	W =  90.000 deg,	P =   0.000 deg,	R =   90.000 deg
};
P[890]{
   GP1:
	UF : 0, UT : 6,		CONFIG : 'N U T, 0, 0, 0',
	X =  218.599  mm,	Y =   -339.634  mm,	Z =   -237.572  mm,
	W =  90.000 deg,	P =   0.000 deg,	R =   90.000 deg
};
P[891]{
   GP1:
	UF : 0, UT : 6,		CONFIG : 'N U T, 0, 0, 0',
	X =  217.772  mm,	Y =   -340.100  mm,	Z =   -237.423  mm,
	W =  90.000 deg,	P =   0.000 deg,	R =   90.000 deg
};
P[892]{
   GP1:
	UF : 0, UT : 6,		CONFIG : 'N U T, 0, 0, 0',
	X =  216.761  mm,	Y =   -340.659  mm,	Z =   -237.124  mm,
	W =  90.000 deg,	P =   0.000 deg,	R =   90.000 deg
};
P[893]{
   GP1:
	UF : 0, UT : 6,		CONFIG : 'N U T, 0, 0, 0',
	X =  216.374  mm,	Y =   -340.918  mm,	Z =   -237.567  mm,
	W =  90.000 deg,	P =   0.000 deg,	R =   90.000 deg
};
P[894]{
   GP1:
	UF : 0, UT : 6,		CONFIG : 'N U T, 0, 0, 0',
	X =  212.724  mm,	Y =   -343.017  mm,	Z =   -237.456  mm,
	W =  90.000 deg,	P =   0.000 deg,	R =   90.000 deg
};
P[895]{
   GP1:
	UF : 0, UT : 6,		CONFIG : 'N U T, 0, 0, 0',
	X =  211.286  mm,	Y =   -343.853  mm,	Z =   -237.533  mm,
	W =  90.000 deg,	P =   0.000 deg,	R =   90.000 deg
};
P[896]{
   GP1:
	UF : 0, UT : 6,		CONFIG : 'N U T, 0, 0, 0',
	X =  210.442  mm,	Y =   -344.341  mm,	Z =   -237.534  mm,
	W =  90.000 deg,	P =   0.000 deg,	R =   90.000 deg
};
P[897]{
   GP1:
	UF : 0, UT : 6,		CONFIG : 'N U T, 0, 0, 0',
	X =  209.616  mm,	Y =   -344.820  mm,	Z =   -237.559  mm,
	W =  90.000 deg,	P =   0.000 deg,	R =   90.000 deg
};
P[898]{
   GP1:
	UF : 0, UT : 6,		CONFIG : 'N U T, 0, 0, 0',
	X =  209.031  mm,	Y =   -345.159  mm,	Z =   -237.581  mm,
	W =  90.000 deg,	P =   0.000 deg,	R =   90.000 deg
};
P[899]{
   GP1:
	UF : 0, UT : 6,		CONFIG : 'N U T, 0, 0, 0',
	X =  208.174  mm,	Y =   -345.643  mm,	Z =   -237.446  mm,
	W =  90.000 deg,	P =   0.000 deg,	R =   90.000 deg
};
P[900]{
   GP1:
	UF : 0, UT : 6,		CONFIG : 'N U T, 0, 0, 0',
	X =  207.552  mm,	Y =   -345.976  mm,	Z =   -237.125  mm,
	W =  90.000 deg,	P =   0.000 deg,	R =   90.000 deg
};
P[901]{
   GP1:
	UF : 0, UT : 6,		CONFIG : 'N U T, 0, 0, 0',
	X =  206.694  mm,	Y =   -346.506  mm,	Z =   -237.541  mm,
	W =  90.000 deg,	P =   0.000 deg,	R =   90.000 deg
};
P[902]{
   GP1:
	UF : 0, UT : 6,		CONFIG : 'N U T, 0, 0, 0',
	X =  205.960  mm,	Y =   -346.930  mm,	Z =   -237.542  mm,
	W =  90.000 deg,	P =   0.000 deg,	R =   90.000 deg
};
P[903]{
   GP1:
	UF : 0, UT : 6,		CONFIG : 'N U T, 0, 0, 0',
	X =  204.545  mm,	Y =   -347.747  mm,	Z =   -237.555  mm,
	W =  90.000 deg,	P =   0.000 deg,	R =   90.000 deg
};
P[904]{
   GP1:
	UF : 0, UT : 6,		CONFIG : 'N U T, 0, 0, 0',
	X =  203.611  mm,	Y =   -348.254  mm,	Z =   -237.149  mm,
	W =  90.000 deg,	P =   0.000 deg,	R =   90.000 deg
};
P[905]{
   GP1:
	UF : 0, UT : 6,		CONFIG : 'N U T, 0, 0, 0',
	X =  203.024  mm,	Y =   -348.627  mm,	Z =   -237.570  mm,
	W =  90.000 deg,	P =   0.000 deg,	R =   90.000 deg
};
P[906]{
   GP1:
	UF : 0, UT : 6,		CONFIG : 'N U T, 0, 0, 0',
	X =  201.031  mm,	Y =   -349.741  mm,	Z =   -237.128  mm,
	W =  90.000 deg,	P =   0.000 deg,	R =   90.000 deg
};
P[907]{
   GP1:
	UF : 0, UT : 6,		CONFIG : 'N U T, 0, 0, 0',
	X =  200.166  mm,	Y =   -350.274  mm,	Z =   -237.539  mm,
	W =  90.000 deg,	P =   0.000 deg,	R =   90.000 deg
};
P[908]{
   GP1:
	UF : 0, UT : 6,		CONFIG : 'N U T, 0, 0, 0',
	X =  199.491  mm,	Y =   -350.660  mm,	Z =   -237.486  mm,
	W =  90.000 deg,	P =   0.000 deg,	R =   90.000 deg
};
P[909]{
   GP1:
	UF : 0, UT : 6,		CONFIG : 'N U T, 0, 0, 0',
	X =  197.725  mm,	Y =   -351.651  mm,	Z =   -237.136  mm,
	W =  90.000 deg,	P =   0.000 deg,	R =   90.000 deg
};
P[910]{
   GP1:
	UF : 0, UT : 6,		CONFIG : 'N U T, 0, 0, 0',
	X =  196.185  mm,	Y =   -351.819  mm,	Z =   -228.207  mm,
	W =  90.000 deg,	P =   0.000 deg,	R =   90.000 deg
};
P[911]{
   GP1:
	UF : 0, UT : 6,		CONFIG : 'N U T, 0, 0, 0',
	X =  195.454  mm,	Y =   -352.239  mm,	Z =   -228.186  mm,
	W =  90.000 deg,	P =   0.000 deg,	R =   90.000 deg
};
P[912]{
   GP1:
	UF : 0, UT : 6,		CONFIG : 'N U T, 0, 0, 0',
	X =  194.680  mm,	Y =   -352.685  mm,	Z =   -228.157  mm,
	W =  90.000 deg,	P =   0.000 deg,	R =   90.000 deg
};
P[913]{
   GP1:
	UF : 0, UT : 6,		CONFIG : 'N U T, 0, 0, 0',
	X =  193.253  mm,	Y =   -353.510  mm,	Z =   -228.179  mm,
	W =  90.000 deg,	P =   0.000 deg,	R =   90.000 deg
};
P[914]{
   GP1:
	UF : 0, UT : 6,		CONFIG : 'N U T, 0, 0, 0',
	X =  190.945  mm,	Y =   -354.840  mm,	Z =   -228.146  mm,
	W =  90.000 deg,	P =   0.000 deg,	R =   90.000 deg
};
P[915]{
   GP1:
	UF : 0, UT : 6,		CONFIG : 'N U T, 0, 0, 0',
	X =  189.476  mm,	Y =   -355.695  mm,	Z =   -228.228  mm,
	W =  90.000 deg,	P =   0.000 deg,	R =   90.000 deg
};
P[916]{
   GP1:
	UF : 0, UT : 6,		CONFIG : 'N U T, 0, 0, 0',
	X =  188.747  mm,	Y =   -356.115  mm,	Z =   -228.220  mm,
	W =  90.000 deg,	P =   0.000 deg,	R =   90.000 deg
};
P[917]{
   GP1:
	UF : 0, UT : 6,		CONFIG : 'N U T, 0, 0, 0',
	X =  188.008  mm,	Y =   -356.536  mm,	Z =   -228.156  mm,
	W =  90.000 deg,	P =   0.000 deg,	R =   90.000 deg
};
P[918]{
   GP1:
	UF : 0, UT : 6,		CONFIG : 'N U T, 0, 0, 0',
	X =  187.424  mm,	Y =   -356.869  mm,	Z =   -228.099  mm,
	W =  90.000 deg,	P =   0.000 deg,	R =   90.000 deg
};
P[919]{
   GP1:
	UF : 0, UT : 6,		CONFIG : 'N U T, 0, 0, 0',
	X =  186.556  mm,	Y =   -357.376  mm,	Z =   -228.173  mm,
	W =  90.000 deg,	P =   0.000 deg,	R =   90.000 deg
};
P[920]{
   GP1:
	UF : 0, UT : 6,		CONFIG : 'N U T, 0, 0, 0',
	X =  185.070  mm,	Y =   -358.240  mm,	Z =   -228.236  mm,
	W =  90.000 deg,	P =   0.000 deg,	R =   90.000 deg
};
P[921]{
   GP1:
	UF : 0, UT : 6,		CONFIG : 'N U T, 0, 0, 0',
	X =  183.550  mm,	Y =   -359.114  mm,	Z =   -228.199  mm,
	W =  90.000 deg,	P =   0.000 deg,	R =   90.000 deg
};
P[922]{
   GP1:
	UF : 0, UT : 6,		CONFIG : 'N U T, 0, 0, 0',
	X =  182.145  mm,	Y =   -359.927  mm,	Z =   -228.216  mm,
	W =  90.000 deg,	P =   0.000 deg,	R =   90.000 deg
};
P[923]{
   GP1:
	UF : 0, UT : 6,		CONFIG : 'N U T, 0, 0, 0',
	X =  180.646  mm,	Y =   -360.783  mm,	Z =   -228.098  mm,
	W =  90.000 deg,	P =   0.000 deg,	R =   90.000 deg
};
P[924]{
   GP1:
	UF : 0, UT : 6,		CONFIG : 'N U T, 0, 0, 0',
	X =  179.919  mm,	Y =   -361.208  mm,	Z =   -228.166  mm,
	W =  90.000 deg,	P =   0.000 deg,	R =   90.000 deg
};
P[925]{
   GP1:
	UF : 0, UT : 6,		CONFIG : 'N U T, 0, 0, 0',
	X =  178.391  mm,	Y =   -362.094  mm,	Z =   -228.205  mm,
	W =  90.000 deg,	P =   0.000 deg,	R =   90.000 deg
};
P[926]{
   GP1:
	UF : 0, UT : 6,		CONFIG : 'N U T, 0, 0, 0',
	X =  177.598  mm,	Y =   -362.550  mm,	Z =   -228.194  mm,
	W =  90.000 deg,	P =   0.000 deg,	R =   90.000 deg
};
P[927]{
   GP1:
	UF : 0, UT : 6,		CONFIG : 'N U T, 0, 0, 0',
	X =  176.920  mm,	Y =   -362.944  mm,	Z =   -228.219  mm,
	W =  90.000 deg,	P =   0.000 deg,	R =   90.000 deg
};
P[928]{
   GP1:
	UF : 0, UT : 6,		CONFIG : 'N U T, 0, 0, 0',
	X =  176.225  mm,	Y =   -363.344  mm,	Z =   -228.207  mm,
	W =  90.000 deg,	P =   0.000 deg,	R =   90.000 deg
};
P[929]{
   GP1:
	UF : 0, UT : 6,		CONFIG : 'N U T, 0, 0, 0',
	X =  174.063  mm,	Y =   -364.588  mm,	Z =   -228.160  mm,
	W =  90.000 deg,	P =   0.000 deg,	R =   90.000 deg
};
P[930]{
   GP1:
	UF : 0, UT : 6,		CONFIG : 'N U T, 0, 0, 0',
	X =  172.581  mm,	Y =   -365.449  mm,	Z =   -228.218  mm,
	W =  90.000 deg,	P =   0.000 deg,	R =   90.000 deg
};
P[931]{
   GP1:
	UF : 0, UT : 6,		CONFIG : 'N U T, 0, 0, 0',
	X =  171.778  mm,	Y =   -365.897  mm,	Z =   -228.031  mm,
	W =  90.000 deg,	P =   0.000 deg,	R =   90.000 deg
};
P[932]{
   GP1:
	UF : 0, UT : 6,		CONFIG : 'N U T, 0, 0, 0',
	X =  170.454  mm,	Y =   -366.676  mm,	Z =   -228.212  mm,
	W =  90.000 deg,	P =   0.000 deg,	R =   90.000 deg
};
P[933]{
   GP1:
	UF : 0, UT : 6,		CONFIG : 'N U T, 0, 0, 0',
	X =  168.940  mm,	Y =   -367.552  mm,	Z =   -228.230  mm,
	W =  90.000 deg,	P =   0.000 deg,	R =   90.000 deg
};
P[934]{
   GP1:
	UF : 0, UT : 6,		CONFIG : 'N U T, 0, 0, 0',
	X =  168.133  mm,	Y =   -368.016  mm,	Z =   -228.209  mm,
	W =  90.000 deg,	P =   0.000 deg,	R =   90.000 deg
};
P[935]{
   GP1:
	UF : 0, UT : 6,		CONFIG : 'N U T, 0, 0, 0',
	X =  166.607  mm,	Y =   -368.891  mm,	Z =   -228.125  mm,
	W =  90.000 deg,	P =   0.000 deg,	R =   90.000 deg
};
P[936]{
   GP1:
	UF : 0, UT : 6,		CONFIG : 'N U T, 0, 0, 0',
	X =  165.799  mm,	Y =   -369.362  mm,	Z =   -228.176  mm,
	W =  90.000 deg,	P =   0.000 deg,	R =   90.000 deg
};
P[937]{
   GP1:
	UF : 0, UT : 6,		CONFIG : 'N U T, 0, 0, 0',
	X =  165.109  mm,	Y =   -369.763  mm,	Z =   -228.216  mm,
	W =  90.000 deg,	P =   0.000 deg,	R =   90.000 deg
};
P[938]{
   GP1:
	UF : 0, UT : 6,		CONFIG : 'N U T, 0, 0, 0',
	X =  164.438  mm,	Y =   -370.147  mm,	Z =   -228.169  mm,
	W =  90.000 deg,	P =   0.000 deg,	R =   90.000 deg
};
P[939]{
   GP1:
	UF : 0, UT : 6,		CONFIG : 'N U T, 0, 0, 0',
	X =  163.639  mm,	Y =   -370.610  mm,	Z =   -228.202  mm,
	W =  90.000 deg,	P =   0.000 deg,	R =   90.000 deg
};
P[940]{
   GP1:
	UF : 0, UT : 6,		CONFIG : 'N U T, 0, 0, 0',
	X =  163.129  mm,	Y =   -370.895  mm,	Z =   -228.083  mm,
	W =  90.000 deg,	P =   0.000 deg,	R =   90.000 deg
};
P[941]{
   GP1:
	UF : 0, UT : 6,		CONFIG : 'N U T, 0, 0, 0',
	X =  159.374  mm,	Y =   -373.071  mm,	Z =   -228.177  mm,
	W =  90.000 deg,	P =   0.000 deg,	R =   90.000 deg
};
P[942]{
   GP1:
	UF : 0, UT : 6,		CONFIG : 'N U T, 0, 0, 0',
	X =  157.164  mm,	Y =   -374.351  mm,	Z =   -228.219  mm,
	W =  90.000 deg,	P =   0.000 deg,	R =   90.000 deg
};
P[943]{
   GP1:
	UF : 0, UT : 6,		CONFIG : 'N U T, 0, 0, 0',
	X =  156.355  mm,	Y =   -374.816  mm,	Z =   -228.197  mm,
	W =  90.000 deg,	P =   0.000 deg,	R =   90.000 deg
};
P[944]{
   GP1:
	UF : 0, UT : 6,		CONFIG : 'N U T, 0, 0, 0',
	X =  155.638  mm,	Y =   -375.233  mm,	Z =   -228.228  mm,
	W =  90.000 deg,	P =   0.000 deg,	R =   90.000 deg
};
P[945]{
   GP1:
	UF : 0, UT : 6,		CONFIG : 'N U T, 0, 0, 0',
	X =  153.508  mm,	Y =   -376.450  mm,	Z =   -228.070  mm,
	W =  90.000 deg,	P =   0.000 deg,	R =   90.000 deg
};
P[946]{
   GP1:
	UF : 0, UT : 6,		CONFIG : 'N U T, 0, 0, 0',
	X =  151.208  mm,	Y =   -377.789  mm,	Z =   -228.208  mm,
	W =  90.000 deg,	P =   0.000 deg,	R =   90.000 deg
};
P[947]{
   GP1:
	UF : 0, UT : 6,		CONFIG : 'N U T, 0, 0, 0',
	X =  150.539  mm,	Y =   -378.176  mm,	Z =   -228.222  mm,
	W =  90.000 deg,	P =   0.000 deg,	R =   90.000 deg
};
P[948]{
   GP1:
	UF : 0, UT : 6,		CONFIG : 'N U T, 0, 0, 0',
	X =  149.740  mm,	Y =   -378.633  mm,	Z =   -228.126  mm,
	W =  90.000 deg,	P =   0.000 deg,	R =   90.000 deg
};
P[949]{
   GP1:
	UF : 0, UT : 6,		CONFIG : 'N U T, 0, 0, 0',
	X =  148.977  mm,	Y =   -379.136  mm,	Z =   -228.227  mm,
	W =  90.000 deg,	P =   0.000 deg,	R =   90.000 deg
};
P[950]{
   GP1:
	UF : 0, UT : 6,		CONFIG : 'N U T, 0, 0, 0',
	X =  148.200  mm,	Y =   -379.722  mm,	Z =   -228.031  mm,
	W =  90.000 deg,	P =   0.000 deg,	R =   90.000 deg
};
P[951]{
   GP1:
	UF : 0, UT : 6,		CONFIG : 'N U T, 0, 0, 0',
	X =  147.266  mm,	Y =   -380.698  mm,	Z =   -228.129  mm,
	W =  90.000 deg,	P =   0.000 deg,	R =   90.000 deg
};
P[952]{
   GP1:
	UF : 0, UT : 6,		CONFIG : 'N U T, 0, 0, 0',
	X =  146.233  mm,	Y =   -382.234  mm,	Z =   -228.093  mm,
	W =  90.000 deg,	P =   0.000 deg,	R =   90.000 deg
};
P[953]{
   GP1:
	UF : 0, UT : 6,		CONFIG : 'N U T, 0, 0, 0',
	X =  146.053  mm,	Y =   -382.678  mm,	Z =   -228.225  mm,
	W =  90.000 deg,	P =   0.000 deg,	R =   90.000 deg
};
P[954]{
   GP1:
	UF : 0, UT : 6,		CONFIG : 'N U T, 0, 0, 0',
	X =  145.808  mm,	Y =   -383.274  mm,	Z =   -228.209  mm,
	W =  90.000 deg,	P =   0.000 deg,	R =   90.000 deg
};
P[955]{
   GP1:
	UF : 0, UT : 6,		CONFIG : 'N U T, 0, 0, 0',
	X =  145.478  mm,	Y =   -384.435  mm,	Z =   -228.097  mm,
	W =  90.000 deg,	P =   0.000 deg,	R =   90.000 deg
};
P[956]{
   GP1:
	UF : 0, UT : 6,		CONFIG : 'N U T, 0, 0, 0',
	X =  145.381  mm,	Y =   -387.073  mm,	Z =   -228.188  mm,
	W =  90.000 deg,	P =   0.000 deg,	R =   90.000 deg
};
P[957]{
   GP1:
	UF : 0, UT : 6,		CONFIG : 'N U T, 0, 0, 0',
	X =  145.443  mm,	Y =   -387.440  mm,	Z =   -228.189  mm,
	W =  90.000 deg,	P =   0.000 deg,	R =   90.000 deg
};
P[958]{
   GP1:
	UF : 0, UT : 6,		CONFIG : 'N U T, 0, 0, 0',
	X =  146.144  mm,	Y =   -389.710  mm,	Z =   -228.125  mm,
	W =  90.000 deg,	P =   0.000 deg,	R =   90.000 deg
};
P[959]{
   GP1:
	UF : 0, UT : 6,		CONFIG : 'N U T, 0, 0, 0',
	X =  146.550  mm,	Y =   -390.502  mm,	Z =   -228.144  mm,
	W =  90.000 deg,	P =   0.000 deg,	R =   90.000 deg
};
P[960]{
   GP1:
	UF : 0, UT : 6,		CONFIG : 'N U T, 0, 0, 0',
	X =  146.942  mm,	Y =   -391.181  mm,	Z =   -228.187  mm,
	W =  90.000 deg,	P =   0.000 deg,	R =   90.000 deg
};
P[961]{
   GP1:
	UF : 0, UT : 6,		CONFIG : 'N U T, 0, 0, 0',
	X =  147.804  mm,	Y =   -392.671  mm,	Z =   -228.212  mm,
	W =  90.000 deg,	P =   0.000 deg,	R =   90.000 deg
};
P[962]{
   GP1:
	UF : 0, UT : 6,		CONFIG : 'N U T, 0, 0, 0',
	X =  148.260  mm,	Y =   -393.458  mm,	Z =   -228.223  mm,
	W =  90.000 deg,	P =   0.000 deg,	R =   90.000 deg
};
P[963]{
   GP1:
	UF : 0, UT : 6,		CONFIG : 'N U T, 0, 0, 0',
	X =  150.818  mm,	Y =   -397.896  mm,	Z =   -228.169  mm,
	W =  90.000 deg,	P =   0.000 deg,	R =   90.000 deg
};
P[964]{
   GP1:
	UF : 0, UT : 6,		CONFIG : 'N U T, 0, 0, 0',
	X =  151.256  mm,	Y =   -398.648  mm,	Z =   -228.215  mm,
	W =  90.000 deg,	P =   0.000 deg,	R =   90.000 deg
};
P[965]{
   GP1:
	UF : 0, UT : 6,		CONFIG : 'N U T, 0, 0, 0',
	X =  151.642  mm,	Y =   -399.327  mm,	Z =   -228.140  mm,
	W =  90.000 deg,	P =   0.000 deg,	R =   90.000 deg
};
P[966]{
   GP1:
	UF : 0, UT : 6,		CONFIG : 'N U T, 0, 0, 0',
	X =  153.792  mm,	Y =   -403.044  mm,	Z =   -228.191  mm,
	W =  90.000 deg,	P =   0.000 deg,	R =   90.000 deg
};
P[967]{
   GP1:
	UF : 0, UT : 6,		CONFIG : 'N U T, 0, 0, 0',
	X =  154.199  mm,	Y =   -403.752  mm,	Z =   -228.164  mm,
	W =  90.000 deg,	P =   0.000 deg,	R =   90.000 deg
};
P[968]{
   GP1:
	UF : 0, UT : 6,		CONFIG : 'N U T, 0, 0, 0',
	X =  154.648  mm,	Y =   -404.525  mm,	Z =   -228.193  mm,
	W =  90.000 deg,	P =   0.000 deg,	R =   90.000 deg
};
P[969]{
   GP1:
	UF : 0, UT : 6,		CONFIG : 'N U T, 0, 0, 0',
	X =  155.420  mm,	Y =   -405.865  mm,	Z =   -228.172  mm,
	W =  90.000 deg,	P =   0.000 deg,	R =   90.000 deg
};
P[970]{
   GP1:
	UF : 0, UT : 6,		CONFIG : 'N U T, 0, 0, 0',
	X =  155.841  mm,	Y =   -406.599  mm,	Z =   -228.138  mm,
	W =  90.000 deg,	P =   0.000 deg,	R =   90.000 deg
};
P[971]{
   GP1:
	UF : 0, UT : 6,		CONFIG : 'N U T, 0, 0, 0',
	X =  157.126  mm,	Y =   -408.820  mm,	Z =   -228.166  mm,
	W =  90.000 deg,	P =   0.000 deg,	R =   90.000 deg
};
P[972]{
   GP1:
	UF : 0, UT : 6,		CONFIG : 'N U T, 0, 0, 0',
	X =  158.080  mm,	Y =   -410.465  mm,	Z =   -228.218  mm,
	W =  90.000 deg,	P =   0.000 deg,	R =   90.000 deg
};
P[973]{
   GP1:
	UF : 0, UT : 6,		CONFIG : 'N U T, 0, 0, 0',
	X =  158.486  mm,	Y =   -411.171  mm,	Z =   -228.203  mm,
	W =  90.000 deg,	P =   0.000 deg,	R =   90.000 deg
};
P[974]{
   GP1:
	UF : 0, UT : 6,		CONFIG : 'N U T, 0, 0, 0',
	X =  158.921  mm,	Y =   -411.930  mm,	Z =   -228.164  mm,
	W =  90.000 deg,	P =   0.000 deg,	R =   90.000 deg
};
P[975]{
   GP1:
	UF : 0, UT : 6,		CONFIG : 'N U T, 0, 0, 0',
	X =  159.712  mm,	Y =   -413.295  mm,	Z =   -228.196  mm,
	W =  90.000 deg,	P =   0.000 deg,	R =   90.000 deg
};
P[976]{
   GP1:
	UF : 0, UT : 6,		CONFIG : 'N U T, 0, 0, 0',
	X =  160.187  mm,	Y =   -414.120  mm,	Z =   -228.194  mm,
	W =  90.000 deg,	P =   0.000 deg,	R =   90.000 deg
};
P[977]{
   GP1:
	UF : 0, UT : 6,		CONFIG : 'N U T, 0, 0, 0',
	X =  160.929  mm,	Y =   -415.417  mm,	Z =   -228.106  mm,
	W =  90.000 deg,	P =   0.000 deg,	R =   90.000 deg
};
P[978]{
   GP1:
	UF : 0, UT : 6,		CONFIG : 'N U T, 0, 0, 0',
	X =  161.858  mm,	Y =   -417.021  mm,	Z =   -228.139  mm,
	W =  90.000 deg,	P =   0.000 deg,	R =   90.000 deg
};
P[979]{
   GP1:
	UF : 0, UT : 6,		CONFIG : 'N U T, 0, 0, 0',
	X =  162.280  mm,	Y =   -417.744  mm,	Z =   -228.199  mm,
	W =  90.000 deg,	P =   0.000 deg,	R =   90.000 deg
};
P[980]{
   GP1:
	UF : 0, UT : 6,		CONFIG : 'N U T, 0, 0, 0',
	X =  162.737  mm,	Y =   -418.529  mm,	Z =   -228.230  mm,
	W =  90.000 deg,	P =   0.000 deg,	R =   90.000 deg
};
P[981]{
   GP1:
	UF : 0, UT : 6,		CONFIG : 'N U T, 0, 0, 0',
	X =  163.999  mm,	Y =   -420.714  mm,	Z =   -228.237  mm,
	W =  90.000 deg,	P =   0.000 deg,	R =   90.000 deg
};
P[982]{
   GP1:
	UF : 0, UT : 6,		CONFIG : 'N U T, 0, 0, 0',
	X =  164.809  mm,	Y =   -422.113  mm,	Z =   -228.236  mm,
	W =  90.000 deg,	P =   0.000 deg,	R =   90.000 deg
};
P[983]{
   GP1:
	UF : 0, UT : 6,		CONFIG : 'N U T, 0, 0, 0',
	X =  165.316  mm,	Y =   -422.912  mm,	Z =   -228.180  mm,
	W =  90.000 deg,	P =   0.000 deg,	R =   90.000 deg
};
P[984]{
   GP1:
	UF : 0, UT : 6,		CONFIG : 'N U T, 0, 0, 0',
	X =  165.883  mm,	Y =   -423.661  mm,	Z =   -228.126  mm,
	W =  90.000 deg,	P =   0.000 deg,	R =   90.000 deg
};
P[985]{
   GP1:
	UF : 0, UT : 6,		CONFIG : 'N U T, 0, 0, 0',
	X =  167.143  mm,	Y =   -424.844  mm,	Z =   -228.228  mm,
	W =  90.000 deg,	P =   0.000 deg,	R =   90.000 deg
};
P[986]{
   GP1:
	UF : 0, UT : 6,		CONFIG : 'N U T, 0, 0, 0',
	X =  167.963  mm,	Y =   -425.401  mm,	Z =   -228.187  mm,
	W =  90.000 deg,	P =   0.000 deg,	R =   90.000 deg
};
P[987]{
   GP1:
	UF : 0, UT : 6,		CONFIG : 'N U T, 0, 0, 0',
	X =  169.627  mm,	Y =   -426.176  mm,	Z =   -228.220  mm,
	W =  90.000 deg,	P =   0.000 deg,	R =   90.000 deg
};
P[988]{
   GP1:
	UF : 0, UT : 6,		CONFIG : 'N U T, 0, 0, 0',
	X =  171.276  mm,	Y =   -426.533  mm,	Z =   -228.200  mm,
	W =  90.000 deg,	P =   0.000 deg,	R =   90.000 deg
};
P[989]{
   GP1:
	UF : 0, UT : 6,		CONFIG : 'N U T, 0, 0, 0',
	X =  173.180  mm,	Y =   -426.560  mm,	Z =   -228.200  mm,
	W =  90.000 deg,	P =   0.000 deg,	R =   90.000 deg
};
P[990]{
   GP1:
	UF : 0, UT : 6,		CONFIG : 'N U T, 0, 0, 0',
	X =  174.290  mm,	Y =   -426.355  mm,	Z =   -228.235  mm,
	W =  90.000 deg,	P =   0.000 deg,	R =   90.000 deg
};
P[991]{
   GP1:
	UF : 0, UT : 6,		CONFIG : 'N U T, 0, 0, 0',
	X =  176.020  mm,	Y =   -425.728  mm,	Z =   -228.224  mm,
	W =  90.000 deg,	P =   0.000 deg,	R =   90.000 deg
};
P[992]{
   GP1:
	UF : 0, UT : 6,		CONFIG : 'N U T, 0, 0, 0',
	X =  176.814  mm,	Y =   -425.317  mm,	Z =   -228.224  mm,
	W =  90.000 deg,	P =   0.000 deg,	R =   90.000 deg
};
P[993]{
   GP1:
	UF : 0, UT : 6,		CONFIG : 'N U T, 0, 0, 0',
	X =  179.687  mm,	Y =   -423.666  mm,	Z =   -228.132  mm,
	W =  90.000 deg,	P =   0.000 deg,	R =   90.000 deg
};
P[994]{
   GP1:
	UF : 0, UT : 6,		CONFIG : 'N U T, 0, 0, 0',
	X =  181.001  mm,	Y =   -422.898  mm,	Z =   -228.235  mm,
	W =  90.000 deg,	P =   0.000 deg,	R =   90.000 deg
};
P[995]{
   GP1:
	UF : 0, UT : 6,		CONFIG : 'N U T, 0, 0, 0',
	X =  183.357  mm,	Y =   -421.546  mm,	Z =   -228.150  mm,
	W =  90.000 deg,	P =   0.000 deg,	R =   90.000 deg
};
P[996]{
   GP1:
	UF : 0, UT : 6,		CONFIG : 'N U T, 0, 0, 0',
	X =  184.091  mm,	Y =   -421.118  mm,	Z =   -228.196  mm,
	W =  90.000 deg,	P =   0.000 deg,	R =   90.000 deg
};
P[997]{
   GP1:
	UF : 0, UT : 6,		CONFIG : 'N U T, 0, 0, 0',
	X =  184.898  mm,	Y =   -420.658  mm,	Z =   -228.123  mm,
	W =  90.000 deg,	P =   0.000 deg,	R =   90.000 deg
};
P[998]{
   GP1:
	UF : 0, UT : 6,		CONFIG : 'N U T, 0, 0, 0',
	X =  186.356  mm,	Y =   -419.822  mm,	Z =   -228.052  mm,
	W =  90.000 deg,	P =   0.000 deg,	R =   90.000 deg
};
P[999]{
   GP1:
	UF : 0, UT : 6,		CONFIG : 'N U T, 0, 0, 0',
	X =  187.838  mm,	Y =   -418.954  mm,	Z =   -228.196  mm,
	W =  90.000 deg,	P =   0.000 deg,	R =   90.000 deg
};
P[1000]{
   GP1:
	UF : 0, UT : 6,		CONFIG : 'N U T, 0, 0, 0',
	X =  189.967  mm,	Y =   -417.730  mm,	Z =   -228.127  mm,
	W =  90.000 deg,	P =   0.000 deg,	R =   90.000 deg
};
P[1001]{
   GP1:
	UF : 0, UT : 6,		CONFIG : 'N U T, 0, 0, 0',
	X =  190.703  mm,	Y =   -417.300  mm,	Z =   -228.188  mm,
	W =  90.000 deg,	P =   0.000 deg,	R =   90.000 deg
};
P[1002]{
   GP1:
	UF : 0, UT : 6,		CONFIG : 'N U T, 0, 0, 0',
	X =  192.914  mm,	Y =   -416.029  mm,	Z =   -228.126  mm,
	W =  90.000 deg,	P =   0.000 deg,	R =   90.000 deg
};
P[1003]{
   GP1:
	UF : 0, UT : 6,		CONFIG : 'N U T, 0, 0, 0',
	X =  193.613  mm,	Y =   -415.619  mm,	Z =   -228.212  mm,
	W =  90.000 deg,	P =   0.000 deg,	R =   90.000 deg
};
P[1004]{
   GP1:
	UF : 0, UT : 6,		CONFIG : 'N U T, 0, 0, 0',
	X =  195.788  mm,	Y =   -414.368  mm,	Z =   -228.146  mm,
	W =  90.000 deg,	P =   0.000 deg,	R =   90.000 deg
};
P[1005]{
   GP1:
	UF : 0, UT : 6,		CONFIG : 'N U T, 0, 0, 0',
	X =  196.586  mm,	Y =   -413.902  mm,	Z =   -228.215  mm,
	W =  90.000 deg,	P =   0.000 deg,	R =   90.000 deg
};
P[1006]{
   GP1:
	UF : 0, UT : 6,		CONFIG : 'N U T, 0, 0, 0',
	X =  197.412  mm,	Y =   -413.423  mm,	Z =   -228.237  mm,
	W =  90.000 deg,	P =   0.000 deg,	R =   90.000 deg
};
P[1007]{
   GP1:
	UF : 0, UT : 6,		CONFIG : 'N U T, 0, 0, 0',
	X =  198.036  mm,	Y =   -413.064  mm,	Z =   -228.228  mm,
	W =  90.000 deg,	P =   0.000 deg,	R =   90.000 deg
};
P[1008]{
   GP1:
	UF : 0, UT : 6,		CONFIG : 'N U T, 0, 0, 0',
	X =  198.778  mm,	Y =   -412.636  mm,	Z =   -228.213  mm,
	W =  90.000 deg,	P =   0.000 deg,	R =   90.000 deg
};
P[1009]{
   GP1:
	UF : 0, UT : 6,		CONFIG : 'N U T, 0, 0, 0',
	X =  200.334  mm,	Y =   -411.737  mm,	Z =   -228.222  mm,
	W =  90.000 deg,	P =   0.000 deg,	R =   90.000 deg
};
P[1010]{
   GP1:
	UF : 0, UT : 6,		CONFIG : 'N U T, 0, 0, 0',
	X =  201.879  mm,	Y =   -410.844  mm,	Z =   -228.237  mm,
	W =  90.000 deg,	P =   0.000 deg,	R =   90.000 deg
};
P[1011]{
   GP1:
	UF : 0, UT : 6,		CONFIG : 'N U T, 0, 0, 0',
	X =  203.269  mm,	Y =   -410.050  mm,	Z =   -228.131  mm,
	W =  90.000 deg,	P =   0.000 deg,	R =   90.000 deg
};
P[1012]{
   GP1:
	UF : 0, UT : 6,		CONFIG : 'N U T, 0, 0, 0',
	X =  205.460  mm,	Y =   -408.780  mm,	Z =   -228.192  mm,
	W =  90.000 deg,	P =   0.000 deg,	R =   90.000 deg
};
P[1013]{
   GP1:
	UF : 0, UT : 6,		CONFIG : 'N U T, 0, 0, 0',
	X =  207.024  mm,	Y =   -407.878  mm,	Z =   -228.181  mm,
	W =  90.000 deg,	P =   0.000 deg,	R =   90.000 deg
};
P[1014]{
   GP1:
	UF : 0, UT : 6,		CONFIG : 'N U T, 0, 0, 0',
	X =  207.746  mm,	Y =   -407.462  mm,	Z =   -228.164  mm,
	W =  90.000 deg,	P =   0.000 deg,	R =   90.000 deg
};
P[1015]{
   GP1:
	UF : 0, UT : 6,		CONFIG : 'N U T, 0, 0, 0',
	X =  209.153  mm,	Y =   -406.651  mm,	Z =   -228.155  mm,
	W =  90.000 deg,	P =   0.000 deg,	R =   90.000 deg
};
P[1016]{
   GP1:
	UF : 0, UT : 6,		CONFIG : 'N U T, 0, 0, 0',
	X =  209.719  mm,	Y =   -406.319  mm,	Z =   -228.208  mm,
	W =  90.000 deg,	P =   0.000 deg,	R =   90.000 deg
};
P[1017]{
   GP1:
	UF : 0, UT : 6,		CONFIG : 'N U T, 0, 0, 0',
	X =  210.677  mm,	Y =   -405.769  mm,	Z =   -228.179  mm,
	W =  90.000 deg,	P =   0.000 deg,	R =   90.000 deg
};
P[1018]{
   GP1:
	UF : 0, UT : 6,		CONFIG : 'N U T, 0, 0, 0',
	X =  211.948  mm,	Y =   -405.031  mm,	Z =   -228.216  mm,
	W =  90.000 deg,	P =   0.000 deg,	R =   90.000 deg
};
P[1019]{
   GP1:
	UF : 0, UT : 6,		CONFIG : 'N U T, 0, 0, 0',
	X =  212.682  mm,	Y =   -404.610  mm,	Z =   -228.190  mm,
	W =  90.000 deg,	P =   0.000 deg,	R =   90.000 deg
};
P[1020]{
   GP1:
	UF : 0, UT : 6,		CONFIG : 'N U T, 0, 0, 0',
	X =  213.487  mm,	Y =   -404.144  mm,	Z =   -228.213  mm,
	W =  90.000 deg,	P =   0.000 deg,	R =   90.000 deg
};
P[1021]{
   GP1:
	UF : 0, UT : 6,		CONFIG : 'N U T, 0, 0, 0',
	X =  215.022  mm,	Y =   -403.262  mm,	Z =   -228.154  mm,
	W =  90.000 deg,	P =   0.000 deg,	R =   90.000 deg
};
P[1022]{
   GP1:
	UF : 0, UT : 6,		CONFIG : 'N U T, 0, 0, 0',
	X =  217.268  mm,	Y =   -401.964  mm,	Z =   -228.169  mm,
	W =  90.000 deg,	P =   0.000 deg,	R =   90.000 deg
};
P[1023]{
   GP1:
	UF : 0, UT : 6,		CONFIG : 'N U T, 0, 0, 0',
	X =  218.082  mm,	Y =   -401.493  mm,	Z =   -228.173  mm,
	W =  90.000 deg,	P =   0.000 deg,	R =   90.000 deg
};
P[1024]{
   GP1:
	UF : 0, UT : 6,		CONFIG : 'N U T, 0, 0, 0',
	X =  218.710  mm,	Y =   -401.132  mm,	Z =   -228.160  mm,
	W =  90.000 deg,	P =   0.000 deg,	R =   90.000 deg
};
P[1025]{
   GP1:
	UF : 0, UT : 6,		CONFIG : 'N U T, 0, 0, 0',
	X =  219.417  mm,	Y =   -400.722  mm,	Z =   -228.177  mm,
	W =  90.000 deg,	P =   0.000 deg,	R =   90.000 deg
};
P[1026]{
   GP1:
	UF : 0, UT : 6,		CONFIG : 'N U T, 0, 0, 0',
	X =  220.998  mm,	Y =   -399.808  mm,	Z =   -228.202  mm,
	W =  90.000 deg,	P =   0.000 deg,	R =   90.000 deg
};
P[1027]{
   GP1:
	UF : 0, UT : 6,		CONFIG : 'N U T, 0, 0, 0',
	X =  222.414  mm,	Y =   -398.991  mm,	Z =   -228.190  mm,
	W =  90.000 deg,	P =   0.000 deg,	R =   90.000 deg
};
P[1028]{
   GP1:
	UF : 0, UT : 6,		CONFIG : 'N U T, 0, 0, 0',
	X =  223.201  mm,	Y =   -398.535  mm,	Z =   -228.206  mm,
	W =  90.000 deg,	P =   0.000 deg,	R =   90.000 deg
};
P[1029]{
   GP1:
	UF : 0, UT : 6,		CONFIG : 'N U T, 0, 0, 0',
	X =  223.860  mm,	Y =   -398.162  mm,	Z =   -228.118  mm,
	W =  90.000 deg,	P =   0.000 deg,	R =   90.000 deg
};
P[1030]{
   GP1:
	UF : 0, UT : 6,		CONFIG : 'N U T, 0, 0, 0',
	X =  224.610  mm,	Y =   -397.722  mm,	Z =   -228.204  mm,
	W =  90.000 deg,	P =   0.000 deg,	R =   90.000 deg
};
P[1031]{
   GP1:
	UF : 0, UT : 6,		CONFIG : 'N U T, 0, 0, 0',
	X =  225.370  mm,	Y =   -397.282  mm,	Z =   -228.218  mm,
	W =  90.000 deg,	P =   0.000 deg,	R =   90.000 deg
};
P[1032]{
   GP1:
	UF : 0, UT : 6,		CONFIG : 'N U T, 0, 0, 0',
	X =  226.172  mm,	Y =   -396.828  mm,	Z =   -228.106  mm,
	W =  90.000 deg,	P =   0.000 deg,	R =   90.000 deg
};
P[1033]{
   GP1:
	UF : 0, UT : 6,		CONFIG : 'N U T, 0, 0, 0',
	X =  226.816  mm,	Y =   -396.457  mm,	Z =   -228.097  mm,
	W =  90.000 deg,	P =   0.000 deg,	R =   90.000 deg
};
P[1034]{
   GP1:
	UF : 0, UT : 6,		CONFIG : 'N U T, 0, 0, 0',
	X =  228.225  mm,	Y =   -395.635  mm,	Z =   -228.203  mm,
	W =  90.000 deg,	P =   0.000 deg,	R =   90.000 deg
};
P[1035]{
   GP1:
	UF : 0, UT : 6,		CONFIG : 'N U T, 0, 0, 0',
	X =  229.019  mm,	Y =   -395.182  mm,	Z =   -228.134  mm,
	W =  90.000 deg,	P =   0.000 deg,	R =   90.000 deg
};
P[1036]{
   GP1:
	UF : 0, UT : 6,		CONFIG : 'N U T, 0, 0, 0',
	X =  232.005  mm,	Y =   -393.450  mm,	Z =   -228.230  mm,
	W =  90.000 deg,	P =   0.000 deg,	R =   90.000 deg
};
P[1037]{
   GP1:
	UF : 0, UT : 6,		CONFIG : 'N U T, 0, 0, 0',
	X =  233.533  mm,	Y =   -392.571  mm,	Z =   -228.184  mm,
	W =  90.000 deg,	P =   0.000 deg,	R =   90.000 deg
};
P[1038]{
   GP1:
	UF : 0, UT : 6,		CONFIG : 'N U T, 0, 0, 0',
	X =  234.936  mm,	Y =   -391.759  mm,	Z =   -228.212  mm,
	W =  90.000 deg,	P =   0.000 deg,	R =   90.000 deg
};
P[1039]{
   GP1:
	UF : 0, UT : 6,		CONFIG : 'N U T, 0, 0, 0',
	X =  235.718  mm,	Y =   -391.307  mm,	Z =   -228.217  mm,
	W =  90.000 deg,	P =   0.000 deg,	R =   90.000 deg
};
P[1040]{
   GP1:
	UF : 0, UT : 6,		CONFIG : 'N U T, 0, 0, 0',
	X =  236.303  mm,	Y =   -390.970  mm,	Z =   -228.207  mm,
	W =  90.000 deg,	P =   0.000 deg,	R =   90.000 deg
};
P[1041]{
   GP1:
	UF : 0, UT : 6,		CONFIG : 'N U T, 0, 0, 0',
	X =  237.830  mm,	Y =   -390.094  mm,	Z =   -228.139  mm,
	W =  90.000 deg,	P =   0.000 deg,	R =   90.000 deg
};
P[1042]{
   GP1:
	UF : 0, UT : 6,		CONFIG : 'N U T, 0, 0, 0',
	X =  239.298  mm,	Y =   -389.238  mm,	Z =   -228.236  mm,
	W =  90.000 deg,	P =   0.000 deg,	R =   90.000 deg
};
P[1043]{
   GP1:
	UF : 0, UT : 6,		CONFIG : 'N U T, 0, 0, 0',
	X =  240.025  mm,	Y =   -388.824  mm,	Z =   -228.163  mm,
	W =  90.000 deg,	P =   0.000 deg,	R =   90.000 deg
};
P[1044]{
   GP1:
	UF : 0, UT : 6,		CONFIG : 'N U T, 0, 0, 0',
	X =  241.569  mm,	Y =   -387.936  mm,	Z =   -228.133  mm,
	W =  90.000 deg,	P =   0.000 deg,	R =   90.000 deg
};
P[1045]{
   GP1:
	UF : 0, UT : 6,		CONFIG : 'N U T, 0, 0, 0',
	X =  242.253  mm,	Y =   -387.541  mm,	Z =   -228.121  mm,
	W =  90.000 deg,	P =   0.000 deg,	R =   90.000 deg
};
P[1046]{
   GP1:
	UF : 0, UT : 6,		CONFIG : 'N U T, 0, 0, 0',
	X =  242.957  mm,	Y =   -387.135  mm,	Z =   -228.115  mm,
	W =  90.000 deg,	P =   0.000 deg,	R =   90.000 deg
};
P[1047]{
   GP1:
	UF : 0, UT : 6,		CONFIG : 'N U T, 0, 0, 0',
	X =  243.734  mm,	Y =   -386.681  mm,	Z =   -228.188  mm,
	W =  90.000 deg,	P =   0.000 deg,	R =   90.000 deg
};
P[1048]{
   GP1:
	UF : 0, UT : 6,		CONFIG : 'N U T, 0, 0, 0',
	X =  244.571  mm,	Y =   -386.197  mm,	Z =   -228.201  mm,
	W =  90.000 deg,	P =   0.000 deg,	R =   90.000 deg
};
P[1049]{
   GP1:
	UF : 0, UT : 6,		CONFIG : 'N U T, 0, 0, 0',
	X =  246.710  mm,	Y =   -384.961  mm,	Z =   -228.208  mm,
	W =  90.000 deg,	P =   0.000 deg,	R =   90.000 deg
};
P[1050]{
   GP1:
	UF : 0, UT : 6,		CONFIG : 'N U T, 0, 0, 0',
	X =  248.052  mm,	Y =   -384.197  mm,	Z =   -228.072  mm,
	W =  90.000 deg,	P =   0.000 deg,	R =   90.000 deg
};
P[1051]{
   GP1:
	UF : 0, UT : 6,		CONFIG : 'N U T, 0, 0, 0',
	X =  248.888  mm,	Y =   -383.706  mm,	Z =   -228.175  mm,
	W =  90.000 deg,	P =   0.000 deg,	R =   90.000 deg
};
P[1052]{
   GP1:
	UF : 0, UT : 6,		CONFIG : 'N U T, 0, 0, 0',
	X =  250.353  mm,	Y =   -382.857  mm,	Z =   -228.217  mm,
	W =  90.000 deg,	P =   0.000 deg,	R =   90.000 deg
};
P[1053]{
   GP1:
	UF : 0, UT : 6,		CONFIG : 'N U T, 0, 0, 0',
	X =  251.853  mm,	Y =   -381.998  mm,	Z =   -228.135  mm,
	W =  90.000 deg,	P =   0.000 deg,	R =   90.000 deg
};
P[1054]{
   GP1:
	UF : 0, UT : 6,		CONFIG : 'N U T, 0, 0, 0',
	X =  252.655  mm,	Y =   -381.527  mm,	Z =   -228.229  mm,
	W =  90.000 deg,	P =   0.000 deg,	R =   90.000 deg
};
P[1055]{
   GP1:
	UF : 0, UT : 6,		CONFIG : 'N U T, 0, 0, 0',
	X =  253.330  mm,	Y =   -381.160  mm,	Z =   -227.949  mm,
	W =  90.000 deg,	P =   0.000 deg,	R =   90.000 deg
};
P[1056]{
   GP1:
	UF : 0, UT : 6,		CONFIG : 'N U T, 0, 0, 0',
	X =  256.261  mm,	Y =   -379.447  mm,	Z =   -228.199  mm,
	W =  90.000 deg,	P =   0.000 deg,	R =   90.000 deg
};
P[1057]{
   GP1:
	UF : 0, UT : 6,		CONFIG : 'N U T, 0, 0, 0',
	X =  257.756  mm,	Y =   -378.581  mm,	Z =   -228.227  mm,
	W =  90.000 deg,	P =   0.000 deg,	R =   90.000 deg
};
P[1058]{
   GP1:
	UF : 0, UT : 6,		CONFIG : 'N U T, 0, 0, 0',
	X =  259.282  mm,	Y =   -377.700  mm,	Z =   -228.233  mm,
	W =  90.000 deg,	P =   0.000 deg,	R =   90.000 deg
};
P[1059]{
   GP1:
	UF : 0, UT : 6,		CONFIG : 'N U T, 0, 0, 0',
	X =  259.920  mm,	Y =   -377.343  mm,	Z =   -228.091  mm,
	W =  90.000 deg,	P =   0.000 deg,	R =   90.000 deg
};
P[1060]{
   GP1:
	UF : 0, UT : 6,		CONFIG : 'N U T, 0, 0, 0',
	X =  262.204  mm,	Y =   -376.025  mm,	Z =   -228.088  mm,
	W =  90.000 deg,	P =   0.000 deg,	R =   90.000 deg
};
P[1061]{
   GP1:
	UF : 0, UT : 6,		CONFIG : 'N U T, 0, 0, 0',
	X =  262.901  mm,	Y =   -375.613  mm,	Z =   -228.204  mm,
	W =  90.000 deg,	P =   0.000 deg,	R =   90.000 deg
};
P[1062]{
   GP1:
	UF : 0, UT : 6,		CONFIG : 'N U T, 0, 0, 0',
	X =  264.412  mm,	Y =   -374.738  mm,	Z =   -228.229  mm,
	W =  90.000 deg,	P =   0.000 deg,	R =   90.000 deg
};
P[1063]{
   GP1:
	UF : 0, UT : 6,		CONFIG : 'N U T, 0, 0, 0',
	X =  265.862  mm,	Y =   -373.911  mm,	Z =   -228.108  mm,
	W =  90.000 deg,	P =   0.000 deg,	R =   90.000 deg
};
P[1064]{
   GP1:
	UF : 0, UT : 6,		CONFIG : 'N U T, 0, 0, 0',
	X =  267.303  mm,	Y =   -373.073  mm,	Z =   -228.176  mm,
	W =  90.000 deg,	P =   0.000 deg,	R =   90.000 deg
};
P[1065]{
   GP1:
	UF : 0, UT : 6,		CONFIG : 'N U T, 0, 0, 0',
	X =  268.078  mm,	Y =   -372.624  mm,	Z =   -228.202  mm,
	W =  90.000 deg,	P =   0.000 deg,	R =   90.000 deg
};
P[1066]{
   GP1:
	UF : 0, UT : 6,		CONFIG : 'N U T, 0, 0, 0',
	X =  269.538  mm,	Y =   -371.782  mm,	Z =   -228.196  mm,
	W =  90.000 deg,	P =   0.000 deg,	R =   90.000 deg
};
P[1067]{
   GP1:
	UF : 0, UT : 6,		CONFIG : 'N U T, 0, 0, 0',
	X =  270.256  mm,	Y =   -371.364  mm,	Z =   -228.230  mm,
	W =  90.000 deg,	P =   0.000 deg,	R =   90.000 deg
};
P[1068]{
   GP1:
	UF : 0, UT : 6,		CONFIG : 'N U T, 0, 0, 0',
	X =  271.689  mm,	Y =   -370.358  mm,	Z =   -228.196  mm,
	W =  90.000 deg,	P =   0.000 deg,	R =   90.000 deg
};
P[1069]{
   GP1:
	UF : 0, UT : 6,		CONFIG : 'N U T, 0, 0, 0',
	X =  272.719  mm,	Y =   -369.306  mm,	Z =   -228.235  mm,
	W =  90.000 deg,	P =   0.000 deg,	R =   90.000 deg
};
P[1070]{
   GP1:
	UF : 0, UT : 6,		CONFIG : 'N U T, 0, 0, 0',
	X =  273.023  mm,	Y =   -368.960  mm,	Z =   -228.082  mm,
	W =  90.000 deg,	P =   0.000 deg,	R =   90.000 deg
};
P[1071]{
   GP1:
	UF : 0, UT : 6,		CONFIG : 'N U T, 0, 0, 0',
	X =  273.704  mm,	Y =   -367.865  mm,	Z =   -228.209  mm,
	W =  90.000 deg,	P =   0.000 deg,	R =   90.000 deg
};
P[1072]{
   GP1:
	UF : 0, UT : 6,		CONFIG : 'N U T, 0, 0, 0',
	X =  274.422  mm,	Y =   -366.020  mm,	Z =   -227.993  mm,
	W =  90.000 deg,	P =   0.000 deg,	R =   90.000 deg
};
P[1073]{
   GP1:
	UF : 0, UT : 6,		CONFIG : 'N U T, 0, 0, 0',
	X =  274.622  mm,	Y =   -364.846  mm,	Z =   -228.129  mm,
	W =  90.000 deg,	P =   0.000 deg,	R =   90.000 deg
};
P[1074]{
   GP1:
	UF : 0, UT : 6,		CONFIG : 'N U T, 0, 0, 0',
	X =  274.671  mm,	Y =   -364.357  mm,	Z =   -228.155  mm,
	W =  90.000 deg,	P =   0.000 deg,	R =   90.000 deg
};
P[1075]{
   GP1:
	UF : 0, UT : 6,		CONFIG : 'N U T, 0, 0, 0',
	X =  274.651  mm,	Y =   -362.902  mm,	Z =   -227.793  mm,
	W =  90.000 deg,	P =   0.000 deg,	R =   90.000 deg
};
P[1076]{
   GP1:
	UF : 0, UT : 6,		CONFIG : 'N U T, 0, 0, 0',
	X =  273.133  mm,	Y =   -358.933  mm,	Z =   -228.065  mm,
	W =  90.000 deg,	P =   0.000 deg,	R =   90.000 deg
};
P[1077]{
   GP1:
	UF : 0, UT : 6,		CONFIG : 'N U T, 0, 0, 0',
	X =  272.654  mm,	Y =   -358.106  mm,	Z =   -228.094  mm,
	W =  90.000 deg,	P =   0.000 deg,	R =   90.000 deg
};
P[1078]{
   GP1:
	UF : 0, UT : 6,		CONFIG : 'N U T, 0, 0, 0',
	X =  271.734  mm,	Y =   -356.528  mm,	Z =   -228.202  mm,
	W =  90.000 deg,	P =   0.000 deg,	R =   90.000 deg
};
P[1079]{
   GP1:
	UF : 0, UT : 6,		CONFIG : 'N U T, 0, 0, 0',
	X =  270.901  mm,	Y =   -355.073  mm,	Z =   -228.110  mm,
	W =  90.000 deg,	P =   0.000 deg,	R =   90.000 deg
};
P[1080]{
   GP1:
	UF : 0, UT : 6,		CONFIG : 'N U T, 0, 0, 0',
	X =  269.220  mm,	Y =   -352.162  mm,	Z =   -228.109  mm,
	W =  90.000 deg,	P =   0.000 deg,	R =   90.000 deg
};
P[1081]{
   GP1:
	UF : 0, UT : 6,		CONFIG : 'N U T, 0, 0, 0',
	X =  268.316  mm,	Y =   -350.596  mm,	Z =   -228.112  mm,
	W =  90.000 deg,	P =   0.000 deg,	R =   90.000 deg
};
P[1082]{
   GP1:
	UF : 0, UT : 6,		CONFIG : 'N U T, 0, 0, 0',
	X =  267.880  mm,	Y =   -349.853  mm,	Z =   -228.196  mm,
	W =  90.000 deg,	P =   0.000 deg,	R =   90.000 deg
};
P[1083]{
   GP1:
	UF : 0, UT : 6,		CONFIG : 'N U T, 0, 0, 0',
	X =  266.276  mm,	Y =   -347.077  mm,	Z =   -228.207  mm,
	W =  90.000 deg,	P =   0.000 deg,	R =   90.000 deg
};
P[1084]{
   GP1:
	UF : 0, UT : 6,		CONFIG : 'N U T, 0, 0, 0',
	X =  264.970  mm,	Y =   -344.811  mm,	Z =   -228.183  mm,
	W =  90.000 deg,	P =   0.000 deg,	R =   90.000 deg
};
P[1085]{
   GP1:
	UF : 0, UT : 6,		CONFIG : 'N U T, 0, 0, 0',
	X =  264.109  mm,	Y =   -343.324  mm,	Z =   -228.218  mm,
	W =  90.000 deg,	P =   0.000 deg,	R =   90.000 deg
};
P[1086]{
   GP1:
	UF : 0, UT : 6,		CONFIG : 'N U T, 0, 0, 0',
	X =  263.609  mm,	Y =   -342.453  mm,	Z =   -228.176  mm,
	W =  90.000 deg,	P =   0.000 deg,	R =   90.000 deg
};
P[1087]{
   GP1:
	UF : 0, UT : 6,		CONFIG : 'N U T, 0, 0, 0',
	X =  262.764  mm,	Y =   -340.968  mm,	Z =   -228.026  mm,
	W =  90.000 deg,	P =   0.000 deg,	R =   90.000 deg
};
P[1088]{
   GP1:
	UF : 0, UT : 6,		CONFIG : 'N U T, 0, 0, 0',
	X =  261.921  mm,	Y =   -339.529  mm,	Z =   -228.166  mm,
	W =  90.000 deg,	P =   0.000 deg,	R =   90.000 deg
};
P[1089]{
   GP1:
	UF : 0, UT : 6,		CONFIG : 'N U T, 0, 0, 0',
	X =  261.450  mm,	Y =   -338.720  mm,	Z =   -228.218  mm,
	W =  90.000 deg,	P =   0.000 deg,	R =   90.000 deg
};
P[1090]{
   GP1:
	UF : 0, UT : 6,		CONFIG : 'N U T, 0, 0, 0',
	X =  261.087  mm,	Y =   -338.092  mm,	Z =   -228.228  mm,
	W =  90.000 deg,	P =   0.000 deg,	R =   90.000 deg
};
P[1091]{
   GP1:
	UF : 0, UT : 6,		CONFIG : 'N U T, 0, 0, 0',
	X =  260.570  mm,	Y =   -337.184  mm,	Z =   -228.131  mm,
	W =  90.000 deg,	P =   0.000 deg,	R =   90.000 deg
};
P[1092]{
   GP1:
	UF : 0, UT : 6,		CONFIG : 'N U T, 0, 0, 0',
	X =  260.251  mm,	Y =   -336.643  mm,	Z =   -228.210  mm,
	W =  90.000 deg,	P =   0.000 deg,	R =   90.000 deg
};
P[1093]{
   GP1:
	UF : 0, UT : 6,		CONFIG : 'N U T, 0, 0, 0',
	X =  259.836  mm,	Y =   -335.912  mm,	Z =   -228.134  mm,
	W =  90.000 deg,	P =   0.000 deg,	R =   90.000 deg
};
P[1094]{
   GP1:
	UF : 0, UT : 6,		CONFIG : 'N U T, 0, 0, 0',
	X =  258.539  mm,	Y =   -333.675  mm,	Z =   -228.189  mm,
	W =  90.000 deg,	P =   0.000 deg,	R =   90.000 deg
};
P[1095]{
   GP1:
	UF : 0, UT : 6,		CONFIG : 'N U T, 0, 0, 0',
	X =  257.696  mm,	Y =   -332.215  mm,	Z =   -228.205  mm,
	W =  90.000 deg,	P =   0.000 deg,	R =   90.000 deg
};
P[1096]{
   GP1:
	UF : 0, UT : 6,		CONFIG : 'N U T, 0, 0, 0',
	X =  256.758  mm,	Y =   -330.587  mm,	Z =   -228.160  mm,
	W =  90.000 deg,	P =   0.000 deg,	R =   90.000 deg
};
P[1097]{
   GP1:
	UF : 0, UT : 6,		CONFIG : 'N U T, 0, 0, 0',
	X =  256.441  mm,	Y =   -330.046  mm,	Z =   -228.236  mm,
	W =  90.000 deg,	P =   0.000 deg,	R =   90.000 deg
};
P[1098]{
   GP1:
	UF : 0, UT : 6,		CONFIG : 'N U T, 0, 0, 0',
	X =  256.018  mm,	Y =   -329.315  mm,	Z =   -228.235  mm,
	W =  90.000 deg,	P =   0.000 deg,	R =   90.000 deg
};
P[1099]{
   GP1:
	UF : 0, UT : 6,		CONFIG : 'N U T, 0, 0, 0',
	X =  255.607  mm,	Y =   -328.601  mm,	Z =   -228.219  mm,
	W =  90.000 deg,	P =   0.000 deg,	R =   90.000 deg
};
P[1100]{
   GP1:
	UF : 0, UT : 6,		CONFIG : 'N U T, 0, 0, 0',
	X =  255.148  mm,	Y =   -327.795  mm,	Z =   -228.118  mm,
	W =  90.000 deg,	P =   0.000 deg,	R =   90.000 deg
};
P[1101]{
   GP1:
	UF : 0, UT : 6,		CONFIG : 'N U T, 0, 0, 0',
	X =  254.688  mm,	Y =   -327.093  mm,	Z =   -228.175  mm,
	W =  90.000 deg,	P =   0.000 deg,	R =   90.000 deg
};
P[1102]{
   GP1:
	UF : 0, UT : 6,		CONFIG : 'N U T, 0, 0, 0',
	X =  254.138  mm,	Y =   -326.372  mm,	Z =   -228.207  mm,
	W =  90.000 deg,	P =   0.000 deg,	R =   90.000 deg
};
P[1103]{
   GP1:
	UF : 0, UT : 6,		CONFIG : 'N U T, 0, 0, 0',
	X =  253.576  mm,	Y =   -325.756  mm,	Z =   -228.066  mm,
	W =  90.000 deg,	P =   0.000 deg,	R =   90.000 deg
};
P[1104]{
   GP1:
	UF : 0, UT : 6,		CONFIG : 'N U T, 0, 0, 0',
	X =  252.655  mm,	Y =   -324.983  mm,	Z =   -228.149  mm,
	W =  90.000 deg,	P =   0.000 deg,	R =   90.000 deg
};
P[1105]{
   GP1:
	UF : 0, UT : 6,		CONFIG : 'N U T, 0, 0, 0',
	X =  252.035  mm,	Y =   -324.600  mm,	Z =   -228.204  mm,
	W =  90.000 deg,	P =   0.000 deg,	R =   90.000 deg
};
P[1106]{
   GP1:
	UF : 0, UT : 6,		CONFIG : 'N U T, 0, 0, 0',
	X =  251.158  mm,	Y =   -324.139  mm,	Z =   -228.169  mm,
	W =  90.000 deg,	P =   0.000 deg,	R =   90.000 deg
};
P[1107]{
   GP1:
	UF : 0, UT : 6,		CONFIG : 'N U T, 0, 0, 0',
	X =  250.497  mm,	Y =   -323.856  mm,	Z =   -228.048  mm,
	W =  90.000 deg,	P =   0.000 deg,	R =   90.000 deg
};
P[1108]{
   GP1:
	UF : 0, UT : 6,		CONFIG : 'N U T, 0, 0, 0',
	X =  249.354  mm,	Y =   -323.554  mm,	Z =   -228.115  mm,
	W =  90.000 deg,	P =   0.000 deg,	R =   90.000 deg
};
P[1109]{
   GP1:
	UF : 0, UT : 6,		CONFIG : 'N U T, 0, 0, 0',
	X =  248.080  mm,	Y =   -323.400  mm,	Z =   -228.218  mm,
	W =  90.000 deg,	P =   0.000 deg,	R =   90.000 deg
};
P[1110]{
   GP1:
	UF : 0, UT : 6,		CONFIG : 'N U T, 0, 0, 0',
	X =  247.380  mm,	Y =   -323.403  mm,	Z =   -228.114  mm,
	W =  90.000 deg,	P =   0.000 deg,	R =   90.000 deg
};
P[1111]{
   GP1:
	UF : 0, UT : 6,		CONFIG : 'N U T, 0, 0, 0',
	X =  246.637  mm,	Y =   -323.466  mm,	Z =   -228.189  mm,
	W =  90.000 deg,	P =   0.000 deg,	R =   90.000 deg
};
P[1112]{
   GP1:
	UF : 0, UT : 6,		CONFIG : 'N U T, 0, 0, 0',
	X =  245.649  mm,	Y =   -323.645  mm,	Z =   -228.144  mm,
	W =  90.000 deg,	P =   0.000 deg,	R =   90.000 deg
};
P[1113]{
   GP1:
	UF : 0, UT : 6,		CONFIG : 'N U T, 0, 0, 0',
	X =  243.852  mm,	Y =   -324.331  mm,	Z =   -228.181  mm,
	W =  90.000 deg,	P =   0.000 deg,	R =   90.000 deg
};
P[1114]{
   GP1:
	UF : 0, UT : 6,		CONFIG : 'N U T, 0, 0, 0',
	X =  241.735  mm,	Y =   -325.520  mm,	Z =   -228.209  mm,
	W =  90.000 deg,	P =   0.000 deg,	R =   90.000 deg
};
P[1115]{
   GP1:
	UF : 0, UT : 6,		CONFIG : 'N U T, 0, 0, 0',
	X =  241.109  mm,	Y =   -325.877  mm,	Z =   -228.162  mm,
	W =  90.000 deg,	P =   0.000 deg,	R =   90.000 deg
};
P[1116]{
   GP1:
	UF : 0, UT : 6,		CONFIG : 'N U T, 0, 0, 0',
	X =  240.465  mm,	Y =   -326.254  mm,	Z =   -228.227  mm,
	W =  90.000 deg,	P =   0.000 deg,	R =   90.000 deg
};
P[1117]{
   GP1:
	UF : 0, UT : 6,		CONFIG : 'N U T, 0, 0, 0',
	X =  239.558  mm,	Y =   -326.769  mm,	Z =   -228.114  mm,
	W =  90.000 deg,	P =   0.000 deg,	R =   90.000 deg
};
P[1118]{
   GP1:
	UF : 0, UT : 6,		CONFIG : 'N U T, 0, 0, 0',
	X =  238.066  mm,	Y =   -327.640  mm,	Z =   -228.238  mm,
	W =  90.000 deg,	P =   0.000 deg,	R =   90.000 deg
};
P[1119]{
   GP1:
	UF : 0, UT : 6,		CONFIG : 'N U T, 0, 0, 0',
	X =  237.327  mm,	Y =   -328.063  mm,	Z =   -228.192  mm,
	W =  90.000 deg,	P =   0.000 deg,	R =   90.000 deg
};
P[1120]{
   GP1:
	UF : 0, UT : 6,		CONFIG : 'N U T, 0, 0, 0',
	X =  235.958  mm,	Y =   -328.854  mm,	Z =   -228.199  mm,
	W =  90.000 deg,	P =   0.000 deg,	R =   90.000 deg
};
P[1121]{
   GP1:
	UF : 0, UT : 6,		CONFIG : 'N U T, 0, 0, 0',
	X =  234.440  mm,	Y =   -329.729  mm,	Z =   -228.183  mm,
	W =  90.000 deg,	P =   0.000 deg,	R =   90.000 deg
};
P[1122]{
   GP1:
	UF : 0, UT : 6,		CONFIG : 'N U T, 0, 0, 0',
	X =  233.520  mm,	Y =   -330.265  mm,	Z =   -228.235  mm,
	W =  90.000 deg,	P =   0.000 deg,	R =   90.000 deg
};
P[1123]{
   GP1:
	UF : 0, UT : 6,		CONFIG : 'N U T, 0, 0, 0',
	X =  232.251  mm,	Y =   -330.992  mm,	Z =   -228.170  mm,
	W =  90.000 deg,	P =   0.000 deg,	R =   90.000 deg
};
P[1124]{
   GP1:
	UF : 0, UT : 6,		CONFIG : 'N U T, 0, 0, 0',
	X =  231.469  mm,	Y =   -331.443  mm,	Z =   -228.156  mm,
	W =  90.000 deg,	P =   0.000 deg,	R =   90.000 deg
};
P[1125]{
   GP1:
	UF : 0, UT : 6,		CONFIG : 'N U T, 0, 0, 0',
	X =  230.815  mm,	Y =   -331.824  mm,	Z =   -228.202  mm,
	W =  90.000 deg,	P =   0.000 deg,	R =   90.000 deg
};
P[1126]{
   GP1:
	UF : 0, UT : 6,		CONFIG : 'N U T, 0, 0, 0',
	X =  230.056  mm,	Y =   -332.259  mm,	Z =   -228.171  mm,
	W =  90.000 deg,	P =   0.000 deg,	R =   90.000 deg
};
P[1127]{
   GP1:
	UF : 0, UT : 6,		CONFIG : 'N U T, 0, 0, 0',
	X =  227.797  mm,	Y =   -333.567  mm,	Z =   -228.216  mm,
	W =  90.000 deg,	P =   0.000 deg,	R =   90.000 deg
};
P[1128]{
   GP1:
	UF : 0, UT : 6,		CONFIG : 'N U T, 0, 0, 0',
	X =  227.004  mm,	Y =   -334.021  mm,	Z =   -228.158  mm,
	W =  90.000 deg,	P =   0.000 deg,	R =   90.000 deg
};
P[1129]{
   GP1:
	UF : 0, UT : 6,		CONFIG : 'N U T, 0, 0, 0',
	X =  225.571  mm,	Y =   -334.849  mm,	Z =   -228.165  mm,
	W =  90.000 deg,	P =   0.000 deg,	R =   90.000 deg
};
P[1130]{
   GP1:
	UF : 0, UT : 6,		CONFIG : 'N U T, 0, 0, 0',
	X =  224.777  mm,	Y =   -335.309  mm,	Z =   -228.191  mm,
	W =  90.000 deg,	P =   0.000 deg,	R =   90.000 deg
};
P[1131]{
   GP1:
	UF : 0, UT : 6,		CONFIG : 'N U T, 0, 0, 0',
	X =  223.482  mm,	Y =   -336.057  mm,	Z =   -228.188  mm,
	W =  90.000 deg,	P =   0.000 deg,	R =   90.000 deg
};
P[1132]{
   GP1:
	UF : 0, UT : 6,		CONFIG : 'N U T, 0, 0, 0',
	X =  222.731  mm,	Y =   -336.484  mm,	Z =   -228.111  mm,
	W =  90.000 deg,	P =   0.000 deg,	R =   90.000 deg
};
P[1133]{
   GP1:
	UF : 0, UT : 6,		CONFIG : 'N U T, 0, 0, 0',
	X =  221.147  mm,	Y =   -337.406  mm,	Z =   -228.191  mm,
	W =  90.000 deg,	P =   0.000 deg,	R =   90.000 deg
};
P[1134]{
   GP1:
	UF : 0, UT : 6,		CONFIG : 'N U T, 0, 0, 0',
	X =  218.952  mm,	Y =   -338.669  mm,	Z =   -228.143  mm,
	W =  90.000 deg,	P =   0.000 deg,	R =   90.000 deg
};
P[1135]{
   GP1:
	UF : 0, UT : 6,		CONFIG : 'N U T, 0, 0, 0',
	X =  217.468  mm,	Y =   -339.528  mm,	Z =   -228.180  mm,
	W =  90.000 deg,	P =   0.000 deg,	R =   90.000 deg
};
P[1136]{
   GP1:
	UF : 0, UT : 6,		CONFIG : 'N U T, 0, 0, 0',
	X =  216.908  mm,	Y =   -339.847  mm,	Z =   -228.118  mm,
	W =  90.000 deg,	P =   0.000 deg,	R =   90.000 deg
};
P[1137]{
   GP1:
	UF : 0, UT : 6,		CONFIG : 'N U T, 0, 0, 0',
	X =  215.232  mm,	Y =   -340.816  mm,	Z =   -228.136  mm,
	W =  90.000 deg,	P =   0.000 deg,	R =   90.000 deg
};
P[1138]{
   GP1:
	UF : 0, UT : 6,		CONFIG : 'N U T, 0, 0, 0',
	X =  214.443  mm,	Y =   -341.276  mm,	Z =   -228.189  mm,
	W =  90.000 deg,	P =   0.000 deg,	R =   90.000 deg
};
P[1139]{
   GP1:
	UF : 0, UT : 6,		CONFIG : 'N U T, 0, 0, 0',
	X =  213.703  mm,	Y =   -341.704  mm,	Z =   -228.189  mm,
	W =  90.000 deg,	P =   0.000 deg,	R =   90.000 deg
};
P[1140]{
   GP1:
	UF : 0, UT : 6,		CONFIG : 'N U T, 0, 0, 0',
	X =  212.985  mm,	Y =   -342.121  mm,	Z =   -228.224  mm,
	W =  90.000 deg,	P =   0.000 deg,	R =   90.000 deg
};
P[1141]{
   GP1:
	UF : 0, UT : 6,		CONFIG : 'N U T, 0, 0, 0',
	X =  211.653  mm,	Y =   -342.889  mm,	Z =   -228.211  mm,
	W =  90.000 deg,	P =   0.000 deg,	R =   90.000 deg
};
P[1142]{
   GP1:
	UF : 0, UT : 6,		CONFIG : 'N U T, 0, 0, 0',
	X =  207.797  mm,	Y =   -345.103  mm,	Z =   -228.052  mm,
	W =  90.000 deg,	P =   0.000 deg,	R =   90.000 deg
};
P[1143]{
   GP1:
	UF : 0, UT : 6,		CONFIG : 'N U T, 0, 0, 0',
	X =  207.124  mm,	Y =   -345.505  mm,	Z =   -228.226  mm,
	W =  90.000 deg,	P =   0.000 deg,	R =   90.000 deg
};
P[1144]{
   GP1:
	UF : 0, UT : 6,		CONFIG : 'N U T, 0, 0, 0',
	X =  205.737  mm,	Y =   -346.303  mm,	Z =   -228.187  mm,
	W =  90.000 deg,	P =   0.000 deg,	R =   90.000 deg
};
P[1145]{
   GP1:
	UF : 0, UT : 6,		CONFIG : 'N U T, 0, 0, 0',
	X =  204.280  mm,	Y =   -347.146  mm,	Z =   -228.212  mm,
	W =  90.000 deg,	P =   0.000 deg,	R =   90.000 deg
};
P[1146]{
   GP1:
	UF : 0, UT : 6,		CONFIG : 'N U T, 0, 0, 0',
	X =  203.547  mm,	Y =   -347.567  mm,	Z =   -228.196  mm,
	W =  90.000 deg,	P =   0.000 deg,	R =   90.000 deg
};
P[1147]{
   GP1:
	UF : 0, UT : 6,		CONFIG : 'N U T, 0, 0, 0',
	X =  201.252  mm,	Y =   -348.892  mm,	Z =   -228.188  mm,
	W =  90.000 deg,	P =   0.000 deg,	R =   90.000 deg
};
P[1148]{
   GP1:
	UF : 0, UT : 6,		CONFIG : 'N U T, 0, 0, 0',
	X =  200.531  mm,	Y =   -349.307  mm,	Z =   -228.158  mm,
	W =  90.000 deg,	P =   0.000 deg,	R =   90.000 deg
};
P[1149]{
   GP1:
	UF : 0, UT : 6,		CONFIG : 'N U T, 0, 0, 0',
	X =  199.010  mm,	Y =   -350.189  mm,	Z =   -228.212  mm,
	W =  90.000 deg,	P =   0.000 deg,	R =   90.000 deg
};
P[1150]{
   GP1:
	UF : 0, UT : 6,		CONFIG : 'N U T, 0, 0, 0',
	X =  197.615  mm,	Y =   -350.991  mm,	Z =   -228.174  mm,
	W =  90.000 deg,	P =   0.000 deg,	R =   90.000 deg
};
P[1151]{
   GP1:
	UF : 0, UT : 6,		CONFIG : 'N U T, 0, 0, 0',
	X =  196.944  mm,	Y =   -351.377  mm,	Z =   -228.150  mm,
	W =  90.000 deg,	P =   0.000 deg,	R =   90.000 deg
};
P[1152]{
   GP1:
	UF : 0, UT : 6,		CONFIG : 'N U T, 0, 0, 0',
	X =  210.000  mm,	Y =   -375.000  mm,	Z =   -250.000  mm,
	W =  90.000 deg,	P =   0.000 deg,	R =   90.000 deg
};
/END
